// TIA Portal V15.1 export
// export: Created 2024-06-21T08:41:24.5997732Z, ExportSetting WithDefaults, DisplayName Totally Integrated Automation Portal, DisplayVersion V15.1 Update 5, DisplayName TIA Portal Openness, DisplayVersion V15.1 Update 5, DisplayName SINAMICS Startdrive Advanced, DisplayVersion V15.1, DisplayName G130, G150, S120, S150, SINAMICS MV, S210, DisplayVersion V15.1, DisplayName G110M, G120, G120C, G120D, G120P, DisplayVersion V15.1, DisplayName STEP 7 Professional, DisplayVersion V15.1 Update 5, DisplayName STEP 7 Safety, DisplayVersion V15.1, DisplayName WinCC Professional, DisplayVersion V15.1 Update 5, DisplayName SIMATIC Visualization Architect, DisplayVersion V15.1
FUNCTION "209230ZS01Safety" : Void   // FC425, FBD
TITLE = 209230ZS01 Safety
{ S7_Optimized_Access := 'FALSE' }
AUTHOR : VCG
FAMILY : Local
NAME : 610
VERSION : 0.1
// stored: AutoNumber false, IsIECCheckEnabled false, SetENOAutomatically False, UDAEnableTagReadback false
   VAR_OUTPUT
      O_AlarmA : Bool;   // Alarm A
      O_AlarmB : Bool;   // Alarm B
      O_AlarmC : Bool;   // Alarm C
      O_AlarmD : Bool;   // Alarm D
      O_AlarmABCondition : Bool;   // Alarms resetable
      H_IAnim : Word;   // Icon Animation
   END_VAR
BEGIN

REGION Network 1: **** 2.1 - Enable Alarms **** 230AS10XS1 Check if dummy plug is ok
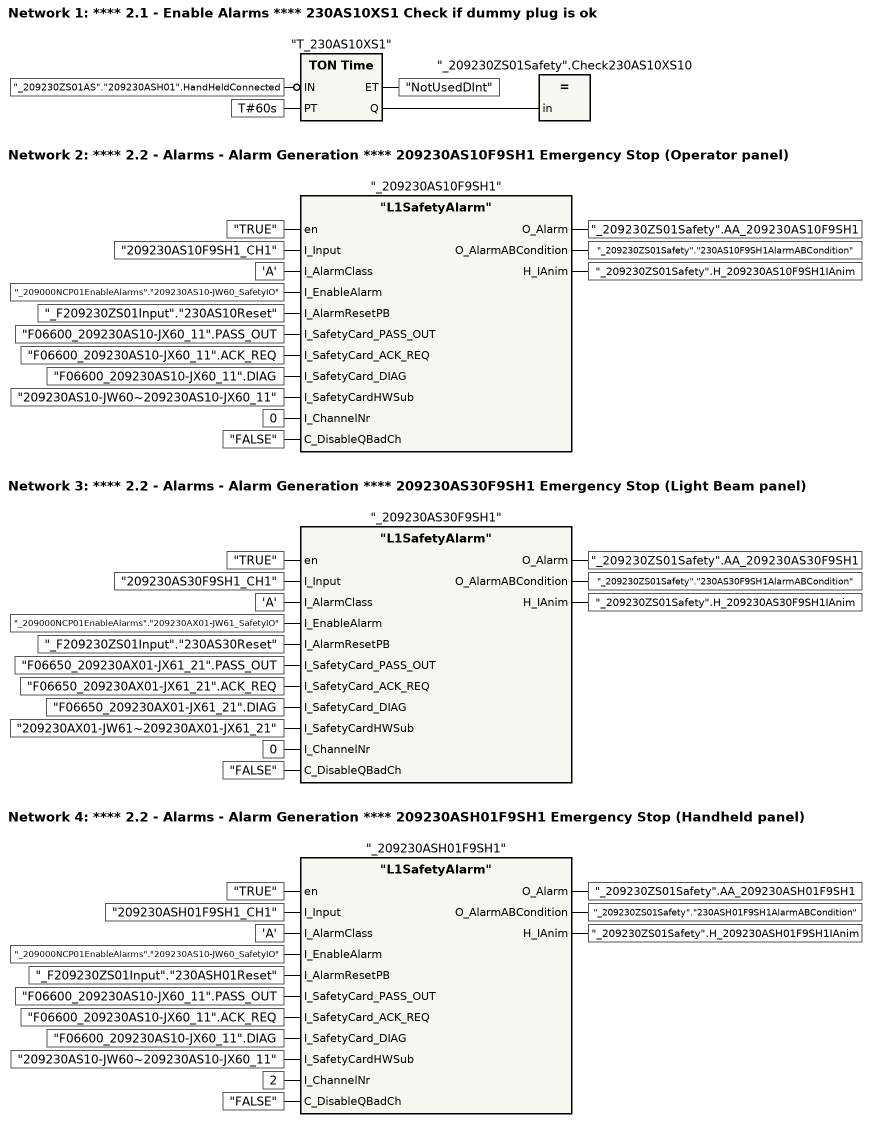
   "T_230AS10XS1".TON(IN := NOT "_209230ZS01AS"."209230ASH01".HandHeldConnected,
                      PT := T#60s,
                      ET => "NotUsedDInt");
   "_209230ZS01Safety".Check230AS10XS10 := "T_230AS10XS1".Q;
END_REGION

REGION Network 2: **** 2.2 - Alarms - Alarm Generation **** 209230AS10F9SH1 Emergency Stop (Operator panel)
   // Emergency Stop
   IF "TRUE" THEN
       "_209230AS10F9SH1"(I_Input := "209230AS10F9SH1_CH1",   // "L1SafetyAlarm"
                          I_AlarmClass := 'A',
                          I_EnableAlarm := "_209000NCP01EnableAlarms"."209230AS10-JW60_SafetyIO",
                          I_AlarmResetPB := "_F209230ZS01Input"."230AS10Reset",
                          I_SafetyCard_PASS_OUT := "F06600_209230AS10-JX60_11".PASS_OUT,
                          I_SafetyCard_ACK_REQ := "F06600_209230AS10-JX60_11".ACK_REQ,
                          I_SafetyCard_DIAG := "F06600_209230AS10-JX60_11".DIAG,
                          I_SafetyCardHWSub := "209230AS10-JW60~209230AS10-JX60_11",
                          I_ChannelNr := 0,
                          C_DisableQBadCh := "FALSE",
                          O_Alarm => "_209230ZS01Safety".AA_209230AS10F9SH1,
                          O_AlarmABCondition => "_209230ZS01Safety"."230AS10F9SH1AlarmABCondition",
                          H_IAnim => "_209230ZS01Safety".H_209230AS10F9SH1IAnim);
   END_IF;
END_REGION

REGION Network 3: **** 2.2 - Alarms - Alarm Generation **** 209230AS30F9SH1 Emergency Stop (Light Beam panel)
   // Emergency Stop
   IF "TRUE" THEN
       "_209230AS30F9SH1"(I_Input := "209230AS30F9SH1_CH1",   // "L1SafetyAlarm"
                          I_AlarmClass := 'A',
                          I_EnableAlarm := "_209000NCP01EnableAlarms"."209230AX01-JW61_SafetyIO",
                          I_AlarmResetPB := "_F209230ZS01Input"."230AS30Reset",
                          I_SafetyCard_PASS_OUT := "F06650_209230AX01-JX61_21".PASS_OUT,
                          I_SafetyCard_ACK_REQ := "F06650_209230AX01-JX61_21".ACK_REQ,
                          I_SafetyCard_DIAG := "F06650_209230AX01-JX61_21".DIAG,
                          I_SafetyCardHWSub := "209230AX01-JW61~209230AX01-JX61_21",
                          I_ChannelNr := 0,
                          C_DisableQBadCh := "FALSE",
                          O_Alarm => "_209230ZS01Safety".AA_209230AS30F9SH1,
                          O_AlarmABCondition => "_209230ZS01Safety"."230AS30F9SH1AlarmABCondition",
                          H_IAnim => "_209230ZS01Safety".H_209230AS30F9SH1IAnim);
   END_IF;
END_REGION

REGION Network 4: **** 2.2 - Alarms - Alarm Generation **** 209230ASH01F9SH1 Emergency Stop (Handheld panel)
   // Emergency Stop
   IF "TRUE" THEN
       "_209230ASH01F9SH1"(I_Input := "209230ASH01F9SH1_CH1",   // "L1SafetyAlarm"
                           I_AlarmClass := 'A',
                           I_EnableAlarm := "_209000NCP01EnableAlarms"."209230AS10-JW60_SafetyIO",
                           I_AlarmResetPB := "_F209230ZS01Input"."230ASH01Reset",
                           I_SafetyCard_PASS_OUT := "F06600_209230AS10-JX60_11".PASS_OUT,
                           I_SafetyCard_ACK_REQ := "F06600_209230AS10-JX60_11".ACK_REQ,
                           I_SafetyCard_DIAG := "F06600_209230AS10-JX60_11".DIAG,
                           I_SafetyCardHWSub := "209230AS10-JW60~209230AS10-JX60_11",
                           I_ChannelNr := 2,
                           C_DisableQBadCh := "FALSE",
                           O_Alarm => "_209230ZS01Safety".AA_209230ASH01F9SH1,
                           O_AlarmABCondition => "_209230ZS01Safety"."230ASH01F9SH1AlarmABCondition",
                           H_IAnim => "_209230ZS01Safety".H_209230ASH01F9SH1IAnim);
   END_IF;
END_REGION

REGION Network 5: **** 2.2 - Alarms - Alarm Generation **** 209230ASD01F9SH1 Emergency Stop (MGB)
   // Emergency Stop
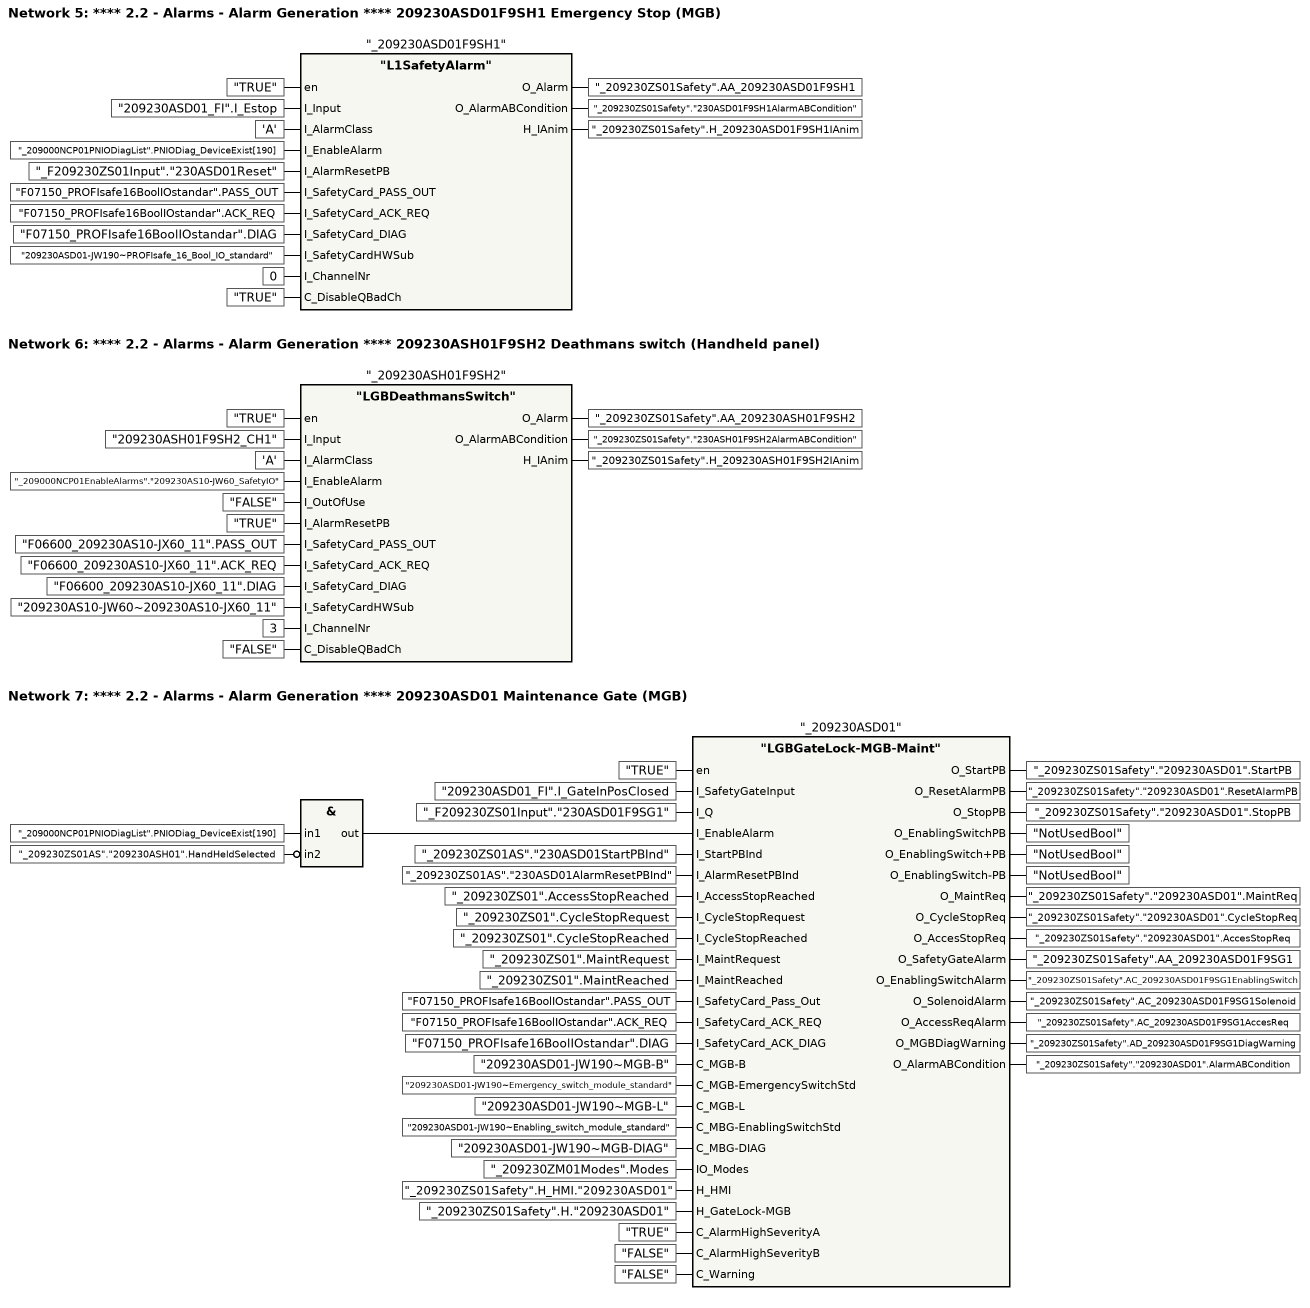
   IF "TRUE" THEN
       "_209230ASD01F9SH1"(I_Input := "209230ASD01_FI".I_Estop,   // "L1SafetyAlarm"
                           I_AlarmClass := 'A',
                           I_EnableAlarm := "_209000NCP01PNIODiagList".PNIODiag_DeviceExist[190],
                           I_AlarmResetPB := "_F209230ZS01Input"."230ASD01Reset",
                           I_SafetyCard_PASS_OUT := "F07150_PROFIsafe16BoolIOstandar".PASS_OUT,
                           I_SafetyCard_ACK_REQ := "F07150_PROFIsafe16BoolIOstandar".ACK_REQ,
                           I_SafetyCard_DIAG := "F07150_PROFIsafe16BoolIOstandar".DIAG,
                           I_SafetyCardHWSub := "209230ASD01-JW190~PROFIsafe_16_Bool_IO_standard",
                           I_ChannelNr := 0,
                           C_DisableQBadCh := "TRUE",
                           O_Alarm => "_209230ZS01Safety".AA_209230ASD01F9SH1,
                           O_AlarmABCondition => "_209230ZS01Safety"."230ASD01F9SH1AlarmABCondition",
                           H_IAnim => "_209230ZS01Safety".H_209230ASD01F9SH1IAnim);
   END_IF;
END_REGION

REGION Network 6: **** 2.2 - Alarms - Alarm Generation **** 209230ASH01F9SH2 Deathmans switch (Handheld panel)
   // Deathmans switch
   IF "TRUE" THEN
       "_209230ASH01F9SH2"(I_Input := "209230ASH01F9SH2_CH1",   // "LGBDeathmansSwitch"
                           I_AlarmClass := 'A',
                           I_EnableAlarm := "_209000NCP01EnableAlarms"."209230AS10-JW60_SafetyIO",
                           I_OutOfUse := "FALSE",
                           I_AlarmResetPB := "TRUE",
                           I_SafetyCard_PASS_OUT := "F06600_209230AS10-JX60_11".PASS_OUT,
                           I_SafetyCard_ACK_REQ := "F06600_209230AS10-JX60_11".ACK_REQ,
                           I_SafetyCard_DIAG := "F06600_209230AS10-JX60_11".DIAG,
                           I_SafetyCardHWSub := "209230AS10-JW60~209230AS10-JX60_11",
                           I_ChannelNr := 3,
                           C_DisableQBadCh := "FALSE",
                           O_Alarm => "_209230ZS01Safety".AA_209230ASH01F9SH2,
                           O_AlarmABCondition => "_209230ZS01Safety"."230ASH01F9SH2AlarmABCondition",
                           H_IAnim => "_209230ZS01Safety".H_209230ASH01F9SH2IAnim);
   END_IF;
END_REGION

REGION Network 7: **** 2.2 - Alarms - Alarm Generation **** 209230ASD01 Maintenance Gate (MGB)
   // Maintenance Gate
   IF "TRUE" THEN
       "_209230ASD01"(I_SafetyGateInput := "209230ASD01_FI".I_GateInPosClosed,   // "LGBGateLock-MGB-Maint"
                      I_Q := "_F209230ZS01Input"."230ASD01F9SG1",
                      I_EnableAlarm := "_209000NCP01PNIODiagList".PNIODiag_DeviceExist[190] AND NOT "_209230ZS01AS"."209230ASH01".HandHeldSelected,
                      I_StartPBInd := "_209230ZS01AS"."230ASD01StartPBInd",
                      I_AlarmResetPBInd := "_209230ZS01AS"."230ASD01AlarmResetPBInd",
                      I_AccessStopReached := "_209230ZS01".AccessStopReached,
                      I_CycleStopRequest := "_209230ZS01".CycleStopRequest,
                      I_CycleStopReached := "_209230ZS01".CycleStopReached,
                      I_MaintRequest := "_209230ZS01".MaintRequest,
                      I_MaintReached := "_209230ZS01".MaintReached,
                      I_SafetyCard_Pass_Out := "F07150_PROFIsafe16BoolIOstandar".PASS_OUT,
                      I_SafetyCard_ACK_REQ := "F07150_PROFIsafe16BoolIOstandar".ACK_REQ,
                      I_SafetyCard_ACK_DIAG := "F07150_PROFIsafe16BoolIOstandar".DIAG,
                      "C_MGB-B" := "209230ASD01-JW190~MGB-B",
                      "C_MGB-EmergencySwitchStd" := "209230ASD01-JW190~Emergency_switch_module_standard",
                      "C_MGB-L" := "209230ASD01-JW190~MGB-L",
                      "C_MBG-EnablingSwitchStd" := "209230ASD01-JW190~Enabling_switch_module_standard",
                      "C_MBG-DIAG" := "209230ASD01-JW190~MGB-DIAG",
                      IO_Modes := "_209230ZM01Modes".Modes,
                      H_HMI := "_209230ZS01Safety".H_HMI."209230ASD01",
                      "H_GateLock-MGB" := "_209230ZS01Safety".H."209230ASD01",
                      C_AlarmHighSeverityA := "TRUE",
                      C_AlarmHighSeverityB := "FALSE",
                      C_Warning := "FALSE",
                      O_StartPB => "_209230ZS01Safety"."209230ASD01".StartPB,
                      O_ResetAlarmPB => "_209230ZS01Safety"."209230ASD01".ResetAlarmPB,
                      O_StopPB => "_209230ZS01Safety"."209230ASD01".StopPB,
                      O_EnablingSwitchPB => "NotUsedBool",
                      "O_EnablingSwitch+PB" => "NotUsedBool",
                      "O_EnablingSwitch-PB" => "NotUsedBool",
                      O_MaintReq => "_209230ZS01Safety"."209230ASD01".MaintReq,
                      O_CycleStopReq => "_209230ZS01Safety"."209230ASD01".CycleStopReq,
                      O_AccesStopReq => "_209230ZS01Safety"."209230ASD01".AccesStopReq,
                      O_SafetyGateAlarm => "_209230ZS01Safety".AA_209230ASD01F9SG1,
                      O_EnablingSwitchAlarm => "_209230ZS01Safety".AC_209230ASD01F9SG1EnablingSwitch,
                      O_SolenoidAlarm => "_209230ZS01Safety".AC_209230ASD01F9SG1Solenoid,
                      O_AccessReqAlarm => "_209230ZS01Safety".AC_209230ASD01F9SG1AccesReq,
                      O_MGBDiagWarning => "_209230ZS01Safety".AD_209230ASD01F9SG1DiagWarning,
                      O_AlarmABCondition => "_209230ZS01Safety"."209230ASD01".AlarmABCondition);
   END_IF;
END_REGION

REGION Network 8: **** 2.2 - Alarms - Alarm Generation **** 209230ZS01F9SG1 Light Curtain
   // Light Curtain
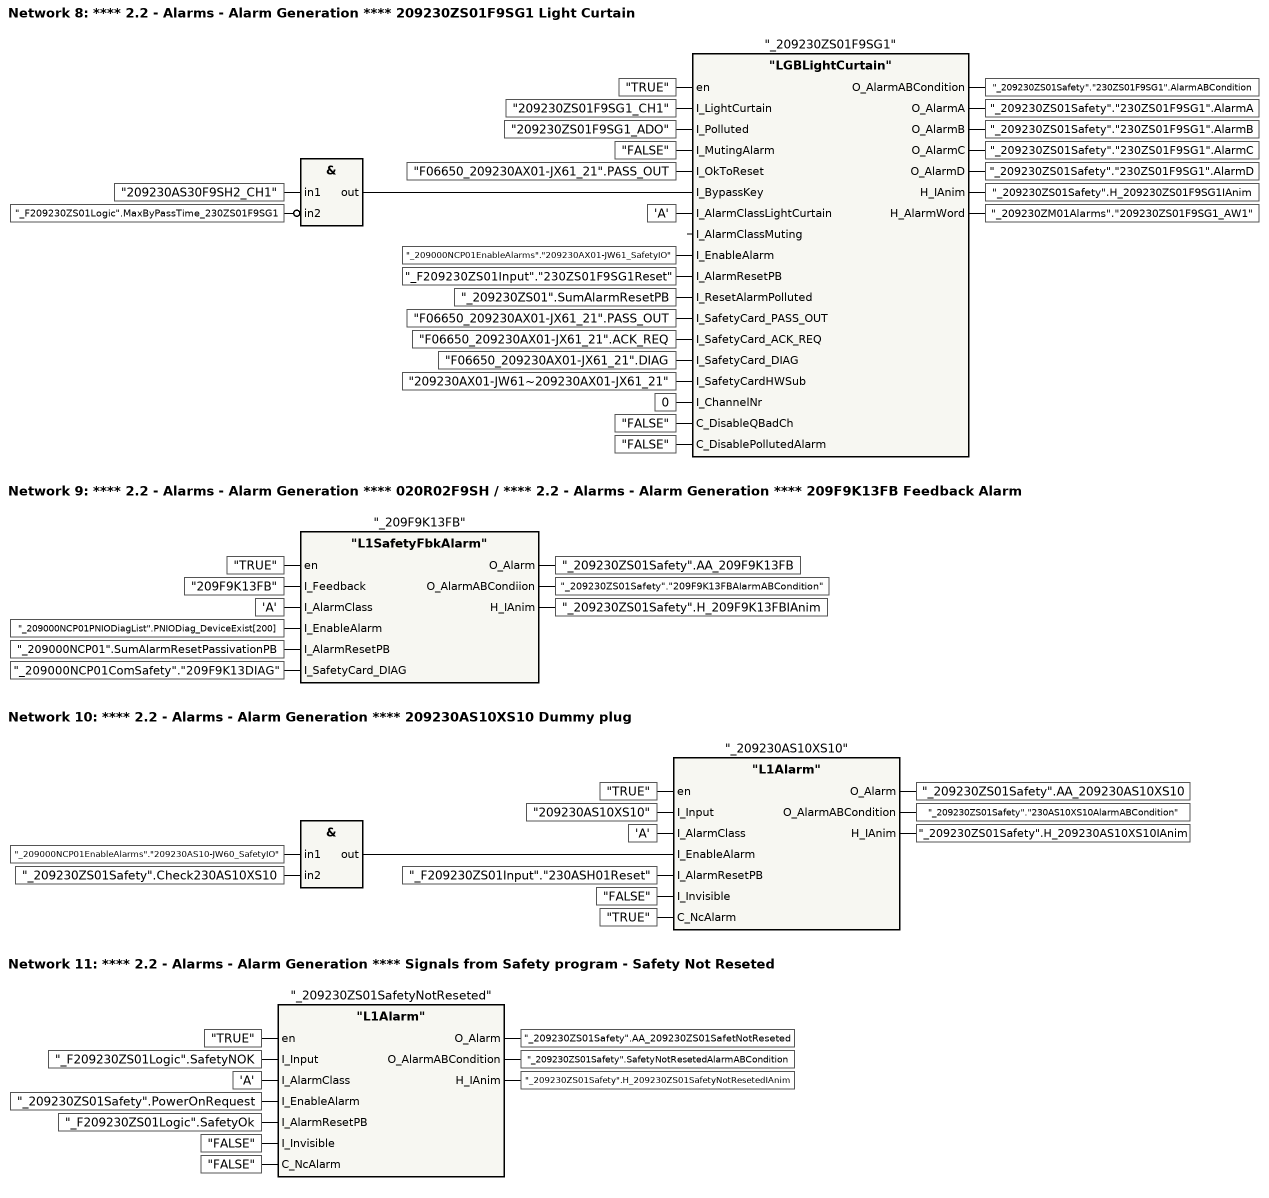
   IF "TRUE" THEN
       "_209230ZS01F9SG1"(I_LightCurtain := "209230ZS01F9SG1_CH1",   // "LGBLightCurtain"
                          I_Polluted := "209230ZS01F9SG1_ADO",
                          I_MutingAlarm := "FALSE",
                          I_OkToReset := "F06650_209230AX01-JX61_21".PASS_OUT,
                          I_BypassKey := "209230AS30F9SH2_CH1" AND NOT "_F209230ZS01Logic".MaxByPassTime_230ZS01F9SG1,
                          I_AlarmClassLightCurtain := 'A',
                          I_EnableAlarm := "_209000NCP01EnableAlarms"."209230AX01-JW61_SafetyIO",
                          I_AlarmResetPB := "_F209230ZS01Input"."230ZS01F9SG1Reset",
                          I_ResetAlarmPolluted := "_209230ZS01".SumAlarmResetPB,
                          I_SafetyCard_PASS_OUT := "F06650_209230AX01-JX61_21".PASS_OUT,
                          I_SafetyCard_ACK_REQ := "F06650_209230AX01-JX61_21".ACK_REQ,
                          I_SafetyCard_DIAG := "F06650_209230AX01-JX61_21".DIAG,
                          I_SafetyCardHWSub := "209230AX01-JW61~209230AX01-JX61_21",
                          I_ChannelNr := 0,
                          C_DisableQBadCh := "FALSE",
                          C_DisablePollutedAlarm := "FALSE",
                          O_AlarmABCondition => "_209230ZS01Safety"."230ZS01F9SG1".AlarmABCondition,
                          O_AlarmA => "_209230ZS01Safety"."230ZS01F9SG1".AlarmA,
                          O_AlarmB => "_209230ZS01Safety"."230ZS01F9SG1".AlarmB,
                          O_AlarmC => "_209230ZS01Safety"."230ZS01F9SG1".AlarmC,
                          O_AlarmD => "_209230ZS01Safety"."230ZS01F9SG1".AlarmD,
                          H_IAnim => "_209230ZS01Safety".H_209230ZS01F9SG1IAnim,
                          H_AlarmWord => "_209230ZM01Alarms"."209230ZS01F9SG1_AW1");
   END_IF;
END_REGION

REGION Network 9: **** 2.2 - Alarms - Alarm Generation **** 020R02F9SH / **** 2.2 - Alarms - Alarm Generation **** 209F9K13FB Feedback Alarm
   // E-Stop Push Button / Feedback Alarm
   IF "TRUE" THEN
       "_209F9K13FB"(I_Feedback := "209F9K13FB",   // "L1SafetyFbkAlarm"
                     I_AlarmClass := 'A',
                     I_EnableAlarm := "_209000NCP01PNIODiagList".PNIODiag_DeviceExist[200],
                     I_AlarmResetPB := "_209000NCP01".SumAlarmResetPassivationPB,
                     I_SafetyCard_DIAG := "_209000NCP01ComSafety"."209F9K13DIAG",
                     O_Alarm => "_209230ZS01Safety".AA_209F9K13FB,
                     O_AlarmABCondiion => "_209230ZS01Safety"."209F9K13FBAlarmABCondition",
                     H_IAnim => "_209230ZS01Safety".H_209F9K13FBIAnim);
   END_IF;
END_REGION

REGION Network 10: **** 2.2 - Alarms - Alarm Generation **** 209230AS10XS10 Dummy plug
   IF "TRUE" THEN
       "_209230AS10XS10"(I_Input := "209230AS10XS10",   // "L1Alarm"
                         I_AlarmClass := 'A',
                         I_EnableAlarm := "_209000NCP01EnableAlarms"."209230AS10-JW60_SafetyIO" AND "_209230ZS01Safety".Check230AS10XS10,
                         I_AlarmResetPB := "_F209230ZS01Input"."230ASH01Reset",
                         I_Invisible := "FALSE",
                         C_NcAlarm := "TRUE",
                         O_Alarm => "_209230ZS01Safety".AA_209230AS10XS10,
                         O_AlarmABCondition => "_209230ZS01Safety"."230AS10XS10AlarmABCondition",
                         H_IAnim => "_209230ZS01Safety".H_209230AS10XS10IAnim);
   END_IF;
END_REGION

REGION Network 11: **** 2.2 - Alarms - Alarm Generation **** Signals from Safety program - Safety Not Reseted
   // Safety Has Not Been Reseted
   IF "TRUE" THEN
       "_209230ZS01SafetyNotReseted"(I_Input := "_F209230ZS01Logic".SafetyNOK,   // "L1Alarm"
                               I_AlarmClass := 'A',
                               I_EnableAlarm := "_209230ZS01Safety".PowerOnRequest,
                               I_AlarmResetPB := "_F209230ZS01Logic".SafetyOk,
                               I_Invisible := "FALSE",
                               C_NcAlarm := "FALSE",
                               O_Alarm => "_209230ZS01Safety".AA_209230ZS01SafetNotReseted,
                               O_AlarmABCondition => "_209230ZS01Safety".SafetyNotResetedAlarmABCondition,
                               H_IAnim => "_209230ZS01Safety".H_209230ZS01SafetyNotResetedIAnim);
   END_IF;
END_REGION

REGION Network 12: **** 2.2 - Alarms - Alarm Generation **** Signals from Safety program - Emergency Stop
   // Emergency Stop
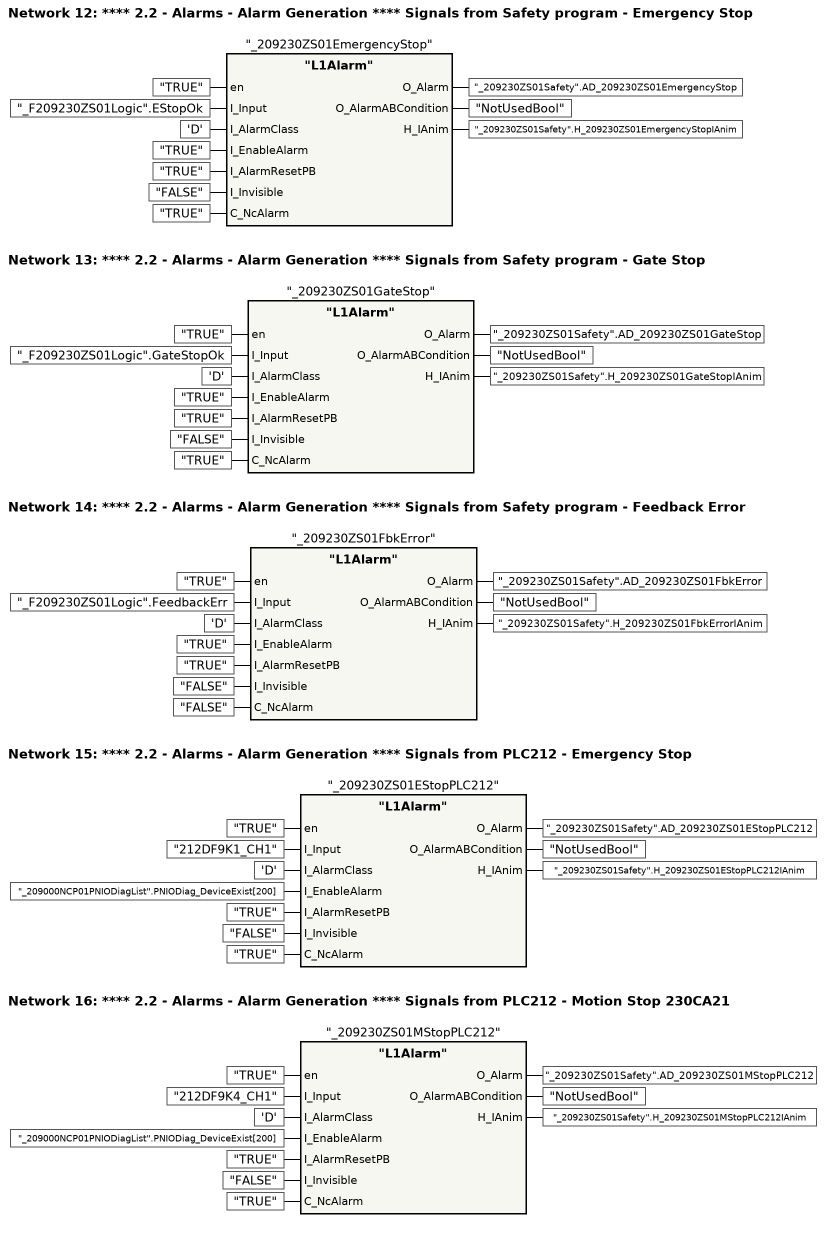
   IF "TRUE" THEN
       "_209230ZS01EmergencyStop"(I_Input := "_F209230ZS01Logic".EStopOk,   // "L1Alarm"
                               I_AlarmClass := 'D',
                               I_EnableAlarm := "TRUE",
                               I_AlarmResetPB := "TRUE",
                               I_Invisible := "FALSE",
                               C_NcAlarm := "TRUE",
                               O_Alarm => "_209230ZS01Safety".AD_209230ZS01EmergencyStop,
                               O_AlarmABCondition => "NotUsedBool",
                               H_IAnim => "_209230ZS01Safety".H_209230ZS01EmergencyStopIAnim);
   END_IF;
END_REGION

REGION Network 13: **** 2.2 - Alarms - Alarm Generation **** Signals from Safety program - Gate Stop
   // Gate Stop
   IF "TRUE" THEN
       "_209230ZS01GateStop"(I_Input := "_F209230ZS01Logic".GateStopOk,   // "L1Alarm"
                             I_AlarmClass := 'D',
                             I_EnableAlarm := "TRUE",
                             I_AlarmResetPB := "TRUE",
                             I_Invisible := "FALSE",
                             C_NcAlarm := "TRUE",
                             O_Alarm => "_209230ZS01Safety".AD_209230ZS01GateStop,
                             O_AlarmABCondition => "NotUsedBool",
                             H_IAnim => "_209230ZS01Safety".H_209230ZS01GateStopIAnim);
   END_IF;
END_REGION

REGION Network 14: **** 2.2 - Alarms - Alarm Generation **** Signals from Safety program - Feedback Error
   // Feedback Error
   IF "TRUE" THEN
       "_209230ZS01FbkError"(I_Input := "_F209230ZS01Logic".FeedbackErr,   // "L1Alarm"
                             I_AlarmClass := 'D',
                             I_EnableAlarm := "TRUE",
                             I_AlarmResetPB := "TRUE",
                             I_Invisible := "FALSE",
                             C_NcAlarm := "FALSE",
                             O_Alarm => "_209230ZS01Safety".AD_209230ZS01FbkError,
                             O_AlarmABCondition => "NotUsedBool",
                             H_IAnim => "_209230ZS01Safety".H_209230ZS01FbkErrorIAnim);
   END_IF;
END_REGION

REGION Network 15: **** 2.2 - Alarms - Alarm Generation **** Signals from PLC212 - Emergency Stop
   IF "TRUE" THEN
       "_209230ZS01EStopPLC212"(I_Input := "212DF9K1_CH1",   // "L1Alarm"
                               I_AlarmClass := 'D',
                               I_EnableAlarm := "_209000NCP01PNIODiagList".PNIODiag_DeviceExist[200],
                               I_AlarmResetPB := "TRUE",
                               I_Invisible := "FALSE",
                               C_NcAlarm := "TRUE",
                               O_Alarm => "_209230ZS01Safety".AD_209230ZS01EStopPLC212,
                               O_AlarmABCondition => "NotUsedBool",
                               H_IAnim => "_209230ZS01Safety".H_209230ZS01EStopPLC212IAnim);
   END_IF;
END_REGION

REGION Network 16: **** 2.2 - Alarms - Alarm Generation **** Signals from PLC212 - Motion Stop 230CA21
   IF "TRUE" THEN
       "_209230ZS01MStopPLC212"(I_Input := "212DF9K4_CH1",   // "L1Alarm"
                               I_AlarmClass := 'D',
                               I_EnableAlarm := "_209000NCP01PNIODiagList".PNIODiag_DeviceExist[200],
                               I_AlarmResetPB := "TRUE",
                               I_Invisible := "FALSE",
                               C_NcAlarm := "TRUE",
                               O_Alarm => "_209230ZS01Safety".AD_209230ZS01MStopPLC212,
                               O_AlarmABCondition => "NotUsedBool",
                               H_IAnim => "_209230ZS01Safety".H_209230ZS01MStopPLC212IAnim);
   END_IF;
END_REGION

REGION Network 17: **** 2.2 - Alarms - Alarm Generation **** Signals from PLC308 - Motion Stop 230CA21
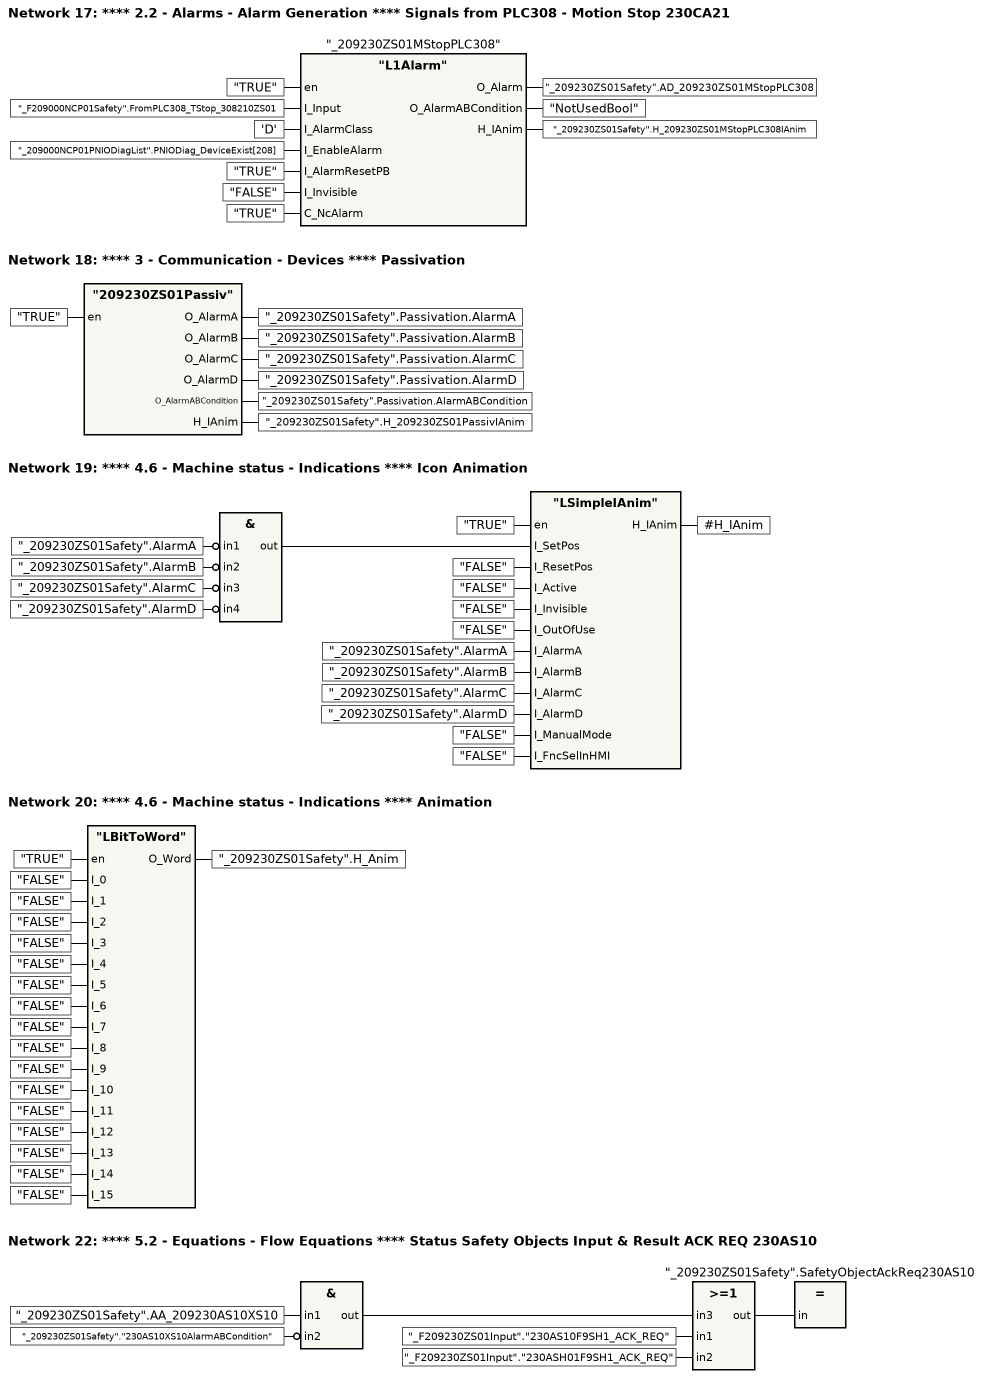
   IF "TRUE" THEN
       "_209230ZS01MStopPLC308"(I_Input := "_F209000NCP01Safety".FromPLC308_TStop_308210ZS01,   // "L1Alarm"
                               I_AlarmClass := 'D',
                               I_EnableAlarm := "_209000NCP01PNIODiagList".PNIODiag_DeviceExist[208],
                               I_AlarmResetPB := "TRUE",
                               I_Invisible := "FALSE",
                               C_NcAlarm := "TRUE",
                               O_Alarm => "_209230ZS01Safety".AD_209230ZS01MStopPLC308,
                               O_AlarmABCondition => "NotUsedBool",
                               H_IAnim => "_209230ZS01Safety".H_209230ZS01MStopPLC308IAnim);
   END_IF;
END_REGION

REGION Network 18: **** 3 - Communication - Devices **** Passivation
   // Passivation
   IF "TRUE" THEN
       "209230ZS01Passiv"(O_AlarmA => "_209230ZS01Safety".Passivation.AlarmA,
                          O_AlarmB => "_209230ZS01Safety".Passivation.AlarmB,
                          O_AlarmC => "_209230ZS01Safety".Passivation.AlarmC,
                          O_AlarmD => "_209230ZS01Safety".Passivation.AlarmD,
                          O_AlarmABCondition => "_209230ZS01Safety".Passivation.AlarmABCondition,
                          H_IAnim => "_209230ZS01Safety".H_209230ZS01PassivIAnim);
   END_IF;
END_REGION

REGION Network 19: **** 4.6 - Machine status - Indications **** Icon Animation
   // Icon animation
   IF "TRUE" THEN
       "LSimpleIAnim"(I_SetPos := NOT "_209230ZS01Safety".AlarmA AND NOT "_209230ZS01Safety".AlarmB AND NOT "_209230ZS01Safety".AlarmC AND NOT "_209230ZS01Safety".AlarmD,
                      I_ResetPos := "FALSE",
                      I_Active := "FALSE",
                      I_Invisible := "FALSE",
                      I_OutOfUse := "FALSE",
                      I_AlarmA := "_209230ZS01Safety".AlarmA,
                      I_AlarmB := "_209230ZS01Safety".AlarmB,
                      I_AlarmC := "_209230ZS01Safety".AlarmC,
                      I_AlarmD := "_209230ZS01Safety".AlarmD,
                      I_ManualMode := "FALSE",
                      I_FncSelInHMI := "FALSE",
                      H_IAnim => #H_IAnim);
   END_IF;
END_REGION

REGION Network 20: **** 4.6 - Machine status - Indications **** Animation
   // Animation
   IF "TRUE" THEN
       "LBitToWord"(I_0 := "FALSE",
                    I_1 := "FALSE",
                    I_2 := "FALSE",
                    I_3 := "FALSE",
                    I_4 := "FALSE",
                    I_5 := "FALSE",
                    I_6 := "FALSE",
                    I_7 := "FALSE",
                    I_8 := "FALSE",
                    I_9 := "FALSE",
                    I_10 := "FALSE",
                    I_11 := "FALSE",
                    I_12 := "FALSE",
                    I_13 := "FALSE",
                    I_14 := "FALSE",
                    I_15 := "FALSE",
                    O_Word => "_209230ZS01Safety".H_Anim);
   END_IF;
END_REGION

NETWORK
TITLE = **** 4.6 - Machine Status - Indications **** Animation DB number
// DB number
      OPN   "_209230ZS01Safety";
      L     DBNO;
      T     "_209230ZS01Safety".H_DBnr;

REGION Network 22: **** 5.2 - Equations - Flow Equations **** Status Safety Objects Input & Result ACK REQ 230AS10
   "_209230ZS01Safety".SafetyObjectAckReq230AS10 := ("_209230ZS01Safety".AA_209230AS10XS10 AND NOT "_209230ZS01Safety"."230AS10XS10AlarmABCondition") OR "_F209230ZS01Input"."230AS10F9SH1_ACK_REQ" OR "_F209230ZS01Input"."230ASH01F9SH1_ACK_REQ";
END_REGION

REGION Network 23: **** 5.2 - Equations - Flow Equations **** Status Safety Objects Input & Result ACK REQ 230AS30
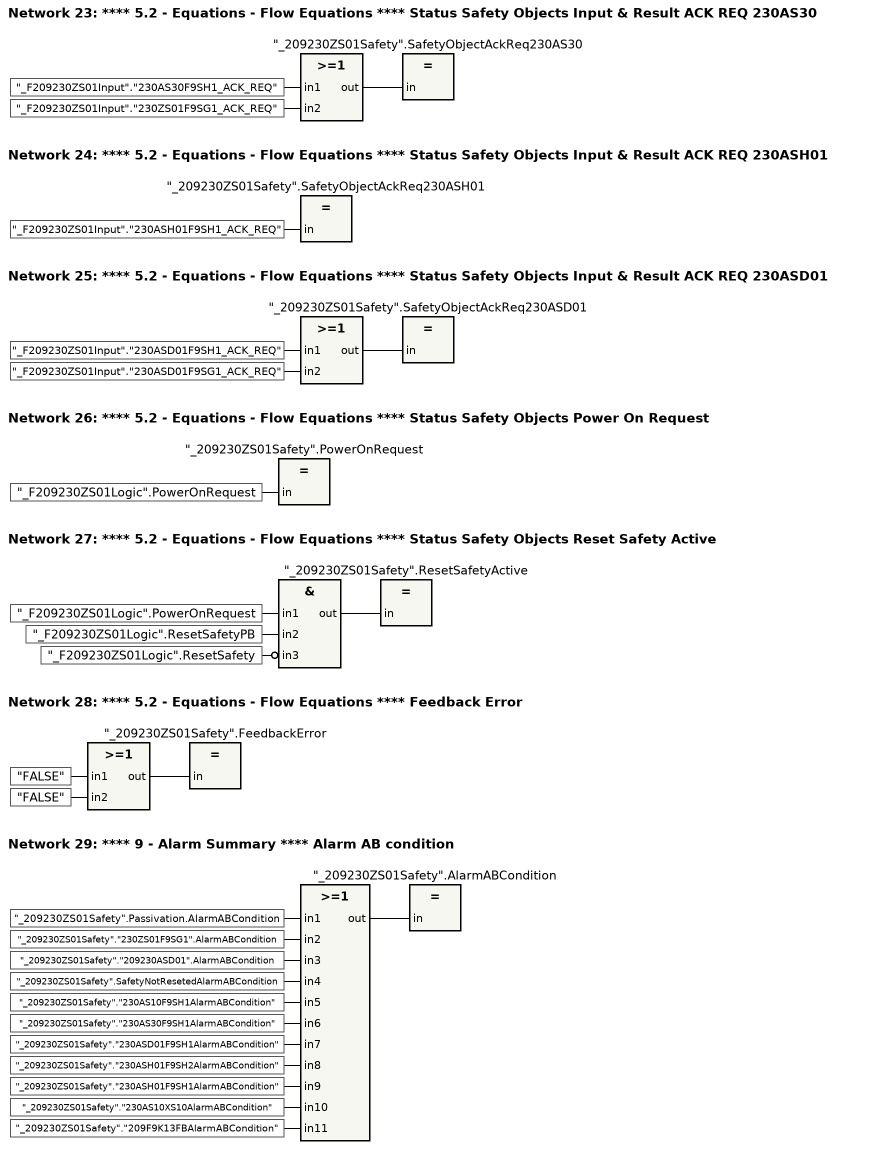
   "_209230ZS01Safety".SafetyObjectAckReq230AS30 := "_F209230ZS01Input"."230AS30F9SH1_ACK_REQ" OR "_F209230ZS01Input"."230ZS01F9SG1_ACK_REQ";
END_REGION

REGION Network 24: **** 5.2 - Equations - Flow Equations **** Status Safety Objects Input & Result ACK REQ 230ASH01
   "_209230ZS01Safety".SafetyObjectAckReq230ASH01 := "_F209230ZS01Input"."230ASH01F9SH1_ACK_REQ";
END_REGION

REGION Network 25: **** 5.2 - Equations - Flow Equations **** Status Safety Objects Input & Result ACK REQ 230ASD01
   "_209230ZS01Safety".SafetyObjectAckReq230ASD01 := "_F209230ZS01Input"."230ASD01F9SH1_ACK_REQ" OR "_F209230ZS01Input"."230ASD01F9SG1_ACK_REQ";
END_REGION

REGION Network 26: **** 5.2 - Equations - Flow Equations **** Status Safety Objects Power On Request
   "_209230ZS01Safety".PowerOnRequest := "_F209230ZS01Logic".PowerOnRequest;
END_REGION

REGION Network 27: **** 5.2 - Equations - Flow Equations **** Status Safety Objects Reset Safety Active
   "_209230ZS01Safety".ResetSafetyActive := "_F209230ZS01Logic".PowerOnRequest AND "_F209230ZS01Logic".ResetSafetyPB AND NOT "_F209230ZS01Logic".ResetSafety;
END_REGION

REGION Network 28: **** 5.2 - Equations - Flow Equations **** Feedback Error
   "_209230ZS01Safety".FeedbackError := "FALSE" OR "FALSE";
END_REGION

REGION Network 29: **** 9 - Alarm Summary **** Alarm AB condition
   // Alarm AB condition
   "_209230ZS01Safety".AlarmABCondition := "_209230ZS01Safety".Passivation.AlarmABCondition OR "_209230ZS01Safety"."230ZS01F9SG1".AlarmABCondition OR "_209230ZS01Safety"."209230ASD01".AlarmABCondition OR "_209230ZS01Safety".SafetyNotResetedAlarmABCondition OR "_209230ZS01Safety"."230AS10F9SH1AlarmABCondition" OR "_209230ZS01Safety"."230AS30F9SH1AlarmABCondition" OR "_209230ZS01Safety"."230ASD01F9SH1AlarmABCondition" OR "_209230ZS01Safety"."230ASH01F9SH2AlarmABCondition" OR "_209230ZS01Safety"."230ASH01F9SH1AlarmABCondition" OR "_209230ZS01Safety"."230AS10XS10AlarmABCondition" OR "_209230ZS01Safety"."209F9K13FBAlarmABCondition";
END_REGION

REGION Network 30: **** 9 - Alarm Summary **** Alarm A
   // Summary of alarms A
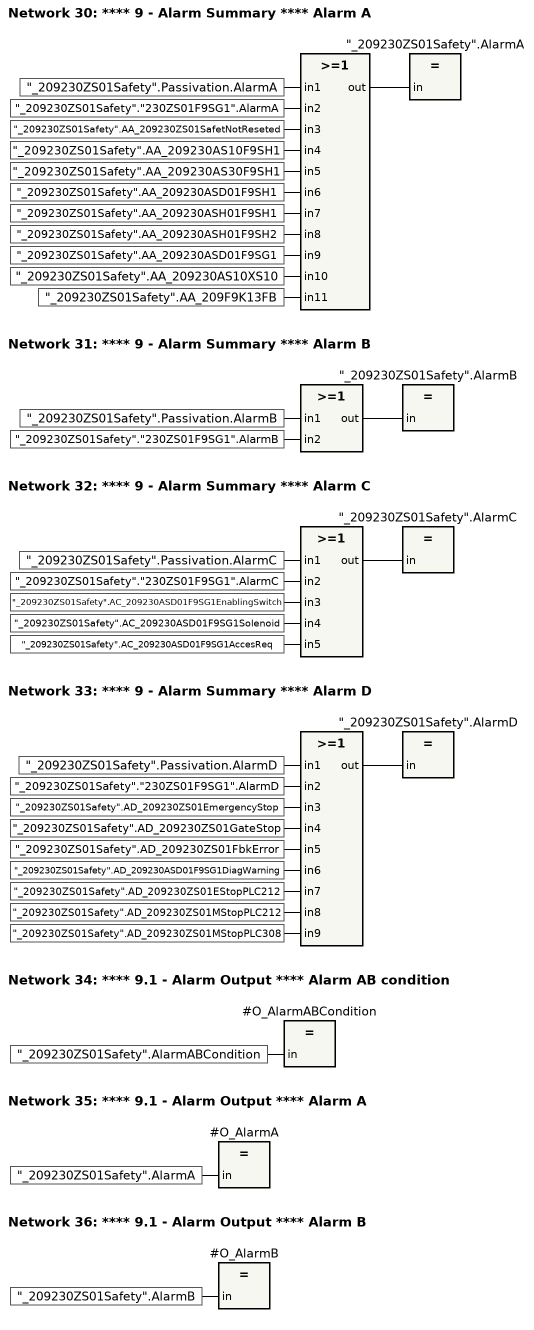
   "_209230ZS01Safety".AlarmA := "_209230ZS01Safety".Passivation.AlarmA OR "_209230ZS01Safety"."230ZS01F9SG1".AlarmA OR "_209230ZS01Safety".AA_209230ZS01SafetNotReseted OR "_209230ZS01Safety".AA_209230AS10F9SH1 OR "_209230ZS01Safety".AA_209230AS30F9SH1 OR "_209230ZS01Safety".AA_209230ASD01F9SH1 OR "_209230ZS01Safety".AA_209230ASH01F9SH1 OR "_209230ZS01Safety".AA_209230ASH01F9SH2 OR "_209230ZS01Safety".AA_209230ASD01F9SG1 OR "_209230ZS01Safety".AA_209230AS10XS10 OR "_209230ZS01Safety".AA_209F9K13FB;
END_REGION

REGION Network 31: **** 9 - Alarm Summary **** Alarm B
   // Summary of alarms B
   "_209230ZS01Safety".AlarmB := "_209230ZS01Safety".Passivation.AlarmB OR "_209230ZS01Safety"."230ZS01F9SG1".AlarmB;
END_REGION

REGION Network 32: **** 9 - Alarm Summary **** Alarm C
   // Summary of alarms C
   "_209230ZS01Safety".AlarmC := "_209230ZS01Safety".Passivation.AlarmC OR "_209230ZS01Safety"."230ZS01F9SG1".AlarmC OR "_209230ZS01Safety".AC_209230ASD01F9SG1EnablingSwitch OR "_209230ZS01Safety".AC_209230ASD01F9SG1Solenoid OR "_209230ZS01Safety".AC_209230ASD01F9SG1AccesReq;
END_REGION

REGION Network 33: **** 9 - Alarm Summary **** Alarm D
   // Summary of alarms D
   "_209230ZS01Safety".AlarmD := "_209230ZS01Safety".Passivation.AlarmD OR "_209230ZS01Safety"."230ZS01F9SG1".AlarmD OR "_209230ZS01Safety".AD_209230ZS01EmergencyStop OR "_209230ZS01Safety".AD_209230ZS01GateStop OR "_209230ZS01Safety".AD_209230ZS01FbkError OR "_209230ZS01Safety".AD_209230ASD01F9SG1DiagWarning OR "_209230ZS01Safety".AD_209230ZS01EStopPLC212 OR "_209230ZS01Safety".AD_209230ZS01MStopPLC212 OR "_209230ZS01Safety".AD_209230ZS01MStopPLC308;
END_REGION

REGION Network 34: **** 9.1 - Alarm Output **** Alarm AB condition
   // Alarm AB condition
   #O_AlarmABCondition := "_209230ZS01Safety".AlarmABCondition;
END_REGION

REGION Network 35: **** 9.1 - Alarm Output **** Alarm A
   // Summary of alarms A
   #O_AlarmA := "_209230ZS01Safety".AlarmA;
END_REGION

REGION Network 36: **** 9.1 - Alarm Output **** Alarm B
   // Summary of alarms B
   #O_AlarmB := "_209230ZS01Safety".AlarmB;
END_REGION

REGION Network 37: **** 9.1 - Alarm Output **** Alarm C
   // Summary of alarms C
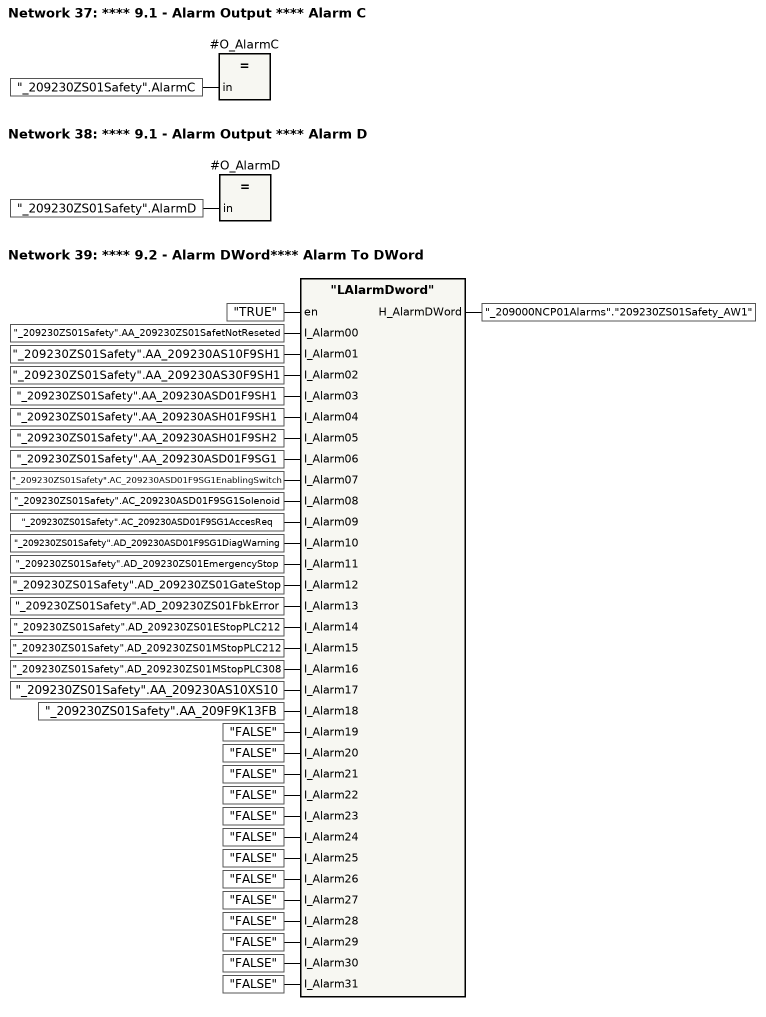
   #O_AlarmC := "_209230ZS01Safety".AlarmC;
END_REGION

REGION Network 38: **** 9.1 - Alarm Output **** Alarm D
   // Summary of alarms D
   #O_AlarmD := "_209230ZS01Safety".AlarmD;
END_REGION

REGION Network 39: **** 9.2 - Alarm DWord**** Alarm To DWord
   // Alarm Word
   IF "TRUE" THEN
       "LAlarmDword"(I_Alarm00 := "_209230ZS01Safety".AA_209230ZS01SafetNotReseted,
                     I_Alarm01 := "_209230ZS01Safety".AA_209230AS10F9SH1,
                     I_Alarm02 := "_209230ZS01Safety".AA_209230AS30F9SH1,
                     I_Alarm03 := "_209230ZS01Safety".AA_209230ASD01F9SH1,
                     I_Alarm04 := "_209230ZS01Safety".AA_209230ASH01F9SH1,
                     I_Alarm05 := "_209230ZS01Safety".AA_209230ASH01F9SH2,
                     I_Alarm06 := "_209230ZS01Safety".AA_209230ASD01F9SG1,
                     I_Alarm07 := "_209230ZS01Safety".AC_209230ASD01F9SG1EnablingSwitch,
                     I_Alarm08 := "_209230ZS01Safety".AC_209230ASD01F9SG1Solenoid,
                     I_Alarm09 := "_209230ZS01Safety".AC_209230ASD01F9SG1AccesReq,
                     I_Alarm10 := "_209230ZS01Safety".AD_209230ASD01F9SG1DiagWarning,
                     I_Alarm11 := "_209230ZS01Safety".AD_209230ZS01EmergencyStop,
                     I_Alarm12 := "_209230ZS01Safety".AD_209230ZS01GateStop,
                     I_Alarm13 := "_209230ZS01Safety".AD_209230ZS01FbkError,
                     I_Alarm14 := "_209230ZS01Safety".AD_209230ZS01EStopPLC212,
                     I_Alarm15 := "_209230ZS01Safety".AD_209230ZS01MStopPLC212,
                     I_Alarm16 := "_209230ZS01Safety".AD_209230ZS01MStopPLC308,
                     I_Alarm17 := "_209230ZS01Safety".AA_209230AS10XS10,
                     I_Alarm18 := "_209230ZS01Safety".AA_209F9K13FB,
                     I_Alarm19 := "FALSE",
                     I_Alarm20 := "FALSE",
                     I_Alarm21 := "FALSE",
                     I_Alarm22 := "FALSE",
                     I_Alarm23 := "FALSE",
                     I_Alarm24 := "FALSE",
                     I_Alarm25 := "FALSE",
                     I_Alarm26 := "FALSE",
                     I_Alarm27 := "FALSE",
                     I_Alarm28 := "FALSE",
                     I_Alarm29 := "FALSE",
                     I_Alarm30 := "FALSE",
                     I_Alarm31 := "FALSE",
                     H_AlarmDWord => "_209000NCP01Alarms"."209230ZS01Safety_AW1");
   END_IF;
END_REGION
END_FUNCTION
